IF NOT (Transfer.Mode = FIT_VFD_Transfer_Modes.Pause) AND NOT (Transfer.Mode = FIT_VFD_Transfer_Modes.Resume) THEN _w1 := Transfer.Mode; END_IF
Transfer.cONFIG.Mode_Memory := _w1;
IF Transfer.Mode = FIT_VFD_Transfer_Modes.Resume THEN _w2 := Transfer.Config.Mode_Memory; END_IF
Transfer.Mode := _w2;
Transfer.Status := SEL(False, SEL(BCV_Not_Ready, SEL(ACV_Not_Ready, SEL(Transfer.Mode=FIT_VFD_Transfer_Modes.Lock_Out, SEL(False, SEL(Complete, SEL(Transfer_Running, SEL(FIT.PLC_Reset, SEL(IDLE_Return, SEL(PAUSED, Transfer_status.IDLE, Transfer_status.Paused), Transfer_status.IDLE), Transfer_status.FIT_Reset), Transfer_status.Running), Transfer_status.Complete), Transfer_status.Complete), Transfer_status.LOCKED_OUT), Transfer_status.ACV_Not_Ready), Transfer_status.BCV_Not_Ready), Transfer_status.VFD_Not_Ready);
_w3 := Transfer.Mode = FIT_VFD_Transfer_Modes.Idle;
_w4 := True AND NOT (BCV.Status = eBCV_Status.A_Closed);
SR2(SET1 := _w3 AND _w4, RESET := NOT _w4); // SR
IF SR2.Q1 THEN _w5 := FIT_VFD_Transfer_Modes.Idle; END_IF
Transfer.Mode := _w5;
BCV_Not_Ready := _w3 AND _w4;
_w6 := 100 - (Transfer.Config.Target_Rate*Transfer.Config.FF);
Transfer.Current_Rate := SEL(Transfer.Config.Active, 0.0, FIT.Rate);
Transfer.Remaining_Time_S := REAL_TO_UDINT(SEL(Transfer_Running, 0.0, Transfer.Remaining_Volume/(Fit.Rate/60)));
_w7 := Transfer.Status = Transfer_Status.Complete;
_w8 := Transfer.Status = Transfer_Status.BCV_Not_Ready OR Transfer.Status = Transfer_Status.VFD_Not_Ready;
_w9 := Transfer_Status.IDLE = Transfer.Status OR False OR Transfer.Status = Transfer_Status.LOCKED_OUT;
_w10 := Transfer.Mode = FIT_VFD_Transfer_Modes.Pause;
PAUSED := _w10;
_w11 := Transfer.Mode = FIT_VFD_Transfer_Modes.IDLE;
_w12 := Complete OR Error OR _w11 OR _w10 OR False;
F_TRIG_0(CLK := Transfer_Running); // F_Trig
TP11(IN := NOT LockOut_Active AND _w12 AND BCV.PLC_CMD, PT := t#1s); // TP
BCV.PLC_CMD := SEL(F_TRIG_0.Q, BCV.PLC_CMD, False);
IDLE_Return := _w8 AND _w11;
SR_10(SET1 := FIT.Total<1, RESET := _w11); // SR
TON_10(IN := SR_10.Q1, PT := T#2s); // TON
FIT_Reset_Complete := TON_10.Q;
R_TRIG_0(CLK := _w11 OR TON_10.Q); // R_trig
_w13 := SEL(R_TRIG_0.Q, FIT.PLC_Reset, False);
_w14 := Transfer.Mode = FIT_VFD_Transfer_Modes.Batch;
_w15 := False OR False OR _w14;
Flow_Mode := _w15;
_w16 := _w15 AND FIT_Reset_Complete AND NOT Complete AND NOT Error AND NOT Time_Complete;
_w17 := _w16 OR (Transfer.Mode=FIT_VFD_Transfer_Modes.Passive);
FT_PIDW_1(
    IN := Transfer.Config.Target_Rate - FIT.Rate,
    KP := Transfer.Config.KP,
    TN := Transfer.Config.TN,
    TV := Transfer.Config.TV,
    LIM_L := 0,
    LIM_H := _w6,
    RST := NOT _w16); // BURKERT_OSCAT_BASIC.FT_PIDW
Transfer.Config.Motor_PCT := SEL(NOT Transfer_Running, LIMIT(0, 100, FT_PIDW_1.Y), 0.0);
Transfer.Config.Active := _w17;
Transfer_Running := _w17;
BCV.PLC_CMD := SEL(_w17, BCV.PLC_CMD, TRUE);
transfer.Remaining_Volume := SEL(_w16, Transfer.Config.Target_Volume, Transfer.Config.Target_Volume-fit.Total);
_w18 := _w14 AND FIT_Reset_Complete AND FIT.Total >= Transfer.Config.Target_Volume;
Batch_Complete := _w18;
RS_11(SET := Time_Complete OR _w18 OR False, RESET1 := _w11); // RS
Complete := RS_11.Q1;
_w19 := LOCK_OUT AND _w9 AND NOT RS_11.Q1;
F_TRIG_10(CLK := _w19); // F_Trig
IF F_TRIG_10.Q THEN _w20 := FIT_VFD_Transfer_Modes.Idle; END_IF
Transfer.Mode := _w20;
_w21 := _w19;
IF _w21 THEN _w22 := FIT_VFD_Transfer_Modes.Lock_Out; END_IF
LockOut_Active := _w21;
Transfer.Mode := _w22;
FIT.PLC_Reset := SEL(NOT SR_10.Q1 AND _w15 AND NOT _w18, _w13, True);
TON_12(IN := _w7, PT := T#30s); // TON
IF TON_12.Q THEN _w23 := FIT_VFD_Transfer_Modes.Idle; END_IF
Transfer.Mode := _w23;
Transfer.Current_Volume := SEL(Transfer.Config.Active, 0.0, FIT.Total);
// Transfer.Mode=FIT_VFD_Transfer_Modes.Passive: input not connected

END_FUNCTION_BLOCK

// 20 Program Organization Units/Transfer_BCV_VFD_FIT_UDFB
FUNCTION_BLOCK Transfer_BCV_VFD_FIT_UDFB
VAR_INPUT
	//Index:INT;
	LOCK_OUT:BOOL:=FALSE;
	
END_VAR
VAR_OUTPUT
END_VAR
VAR
	Paused:BOOL;
	Idle_return:BOOL;
	Transfer_Running:BOOL;
	Complete:BOOL;
	ACV_Not_Ready:BOOL;
	VFD_Not_Ready:BOOL;
	BCV_Not_Ready:BOOL;
	Time_Complete:BOOL;
	FIT_Reset_Complete:BOOL;
	Pump_Start:BOOL;
	Lockout_Active:BOOL;
	Error:BOOL;
	Flow_Mode:BOOL;
	Batch_Complete:BOOL;
	Enable_pump:BOOL;
	
	PID_CV:REAL;
	
	
	
	
	SR2: SR;
	TON_0: TON;
	CTRL_PID_1: BURKERT_OSCAT_BASIC.CTRL_PID;
	R_TRIG_0: R_trig;
	TON_10: TON;
	SR_10: SR;
	RS_11: RS;
	TON_12: TON;
	F_TRIG_10: F_Trig;
	TP11: TP;
	F_TRIG_0: F_Trig;
END_VAR

VAR_IN_OUT
	Transfer:FIT_VFD_Transfer_DUT;
	VFD:VFD_Vacon_DUT;
	BCV:BCV_DUT;
	FIT:FIT_DUT;
	
END_VAR
VAR // added by the converter: edge detectors and wires of the graphical bodies
    _w1, _w2, _w7, _w22, _w24 : ANY;
    _w3, _w4, _w5, _w6, _w8, _w9, _w10, _w11, _w12, _w13, _w14, _w15, _w16, _w17, _w18, _w19, _w20, _w21, _w23, _w25 : BOOL;
    _w26 : REAL;
END_VAR

IF NOT (Transfer.Mode = FIT_VFD_Transfer_Modes.Pause) AND NOT (Transfer.Mode = FIT_VFD_Transfer_Modes.Resume) THEN _w1 := Transfer.Mode; END_IF
Transfer.cONFIG.Mode_Memory := _w1;
IF Transfer.Mode = FIT_VFD_Transfer_Modes.Resume THEN _w2 := Transfer.Config.Mode_Memory; END_IF
Transfer.Mode := _w2;
Transfer.Status := SEL(VFD_Not_Ready, SEL(BCV_Not_Ready, SEL(ACV_Not_Ready, SEL(Transfer.Mode=FIT_VFD_Transfer_Modes.Lock_Out, SEL(False, SEL(Complete, SEL(Transfer_Running, SEL(FIT.PLC_Reset, SEL(IDLE_Return, SEL(PAUSED, Transfer_status.IDLE, Transfer_status.Paused), Transfer_status.IDLE), Transfer_status.FIT_Reset), Transfer_status.Running), Transfer_status.Complete), Transfer_status.Complete), Transfer_status.LOCKED_OUT), Transfer_status.ACV_Not_Ready), Transfer_status.BCV_Not_Ready), Transfer_status.VFD_Not_Ready);
_w3 := Transfer.Mode = FIT_VFD_Transfer_Modes.Idle;
_w4 := True AND NOT (BCV.Status = eBCV_Status.A_Closed);
BCV_Not_Ready := _w3 AND _w4;
_w5 := True AND NOT (VFD.MODE.eMode = VFD_Modes.Auto);
_w6 := _w4 OR _w5;
SR2(SET1 := _w3 AND _w6, RESET := NOT _w6); // SR
IF SR2.Q1 THEN _w7 := FIT_VFD_Transfer_Modes.Idle; END_IF
Transfer.Mode := _w7;
VFD_Not_Ready := _w3 AND _w5;
_w8 := Transfer.Status = Transfer_Status.Complete;
_w9 := Transfer.Status = Transfer_Status.BCV_Not_Ready OR Transfer.Status = Transfer_Status.VFD_Not_Ready;
_w10 := Transfer_Status.IDLE = Transfer.Status OR False OR Transfer.Status = Transfer_Status.LOCKED_OUT;
_w11 := Transfer.Mode = FIT_VFD_Transfer_Modes.Pause;
PAUSED := _w11;
_w12 := Transfer.Mode = FIT_VFD_Transfer_Modes.IDLE;
_w13 := Complete OR Error OR _w12 OR _w11;
_w14 := NOT Pump_Start OR _w13;
CTRL_PID_1(
    ACT := FIT.Rate,
    SET := Transfer.Config.Target_Rate,
    SUP := 0.0,
    OFS := Transfer.Config.Target_Rate * Transfer.Config.FF,
    M_I := 0.0,
    MAN := _w14,
    RST := _w14,
    KP := Transfer.Config.KP,
    TN := Transfer.Config.TN,
    TV := Transfer.Config.TV,
    LL := 0,
    LH := 100); // BURKERT_OSCAT_BASIC.CTRL_PID
PID_CV := CTRL_PID_1.Y;
TP11(IN := NOT LockOut_Active AND _w13, PT := t#5s); // TP
VFD.PLC_Run := SEL(TP11.Q, VFD.PLC_Run, FALSE);
VFD.PLC_CMD := SEL(TP11.Q, VFD.PLC_CMD, 0.0);
F_TRIG_0(CLK := TP11.Q); // F_Trig
BCV.PLC_CMD := SEL(F_TRIG_0.Q, BCV.PLC_CMD, False);
IDLE_Return := _w9 AND _w12;
SR_10(SET1 := FIT.Total<1, RESET := _w12); // SR
TON_10(IN := SR_10.Q1, PT := T#2s); // TON
FIT_Reset_Complete := TON_10.Q;
R_TRIG_0(CLK := _w12 OR TON_10.Q); // R_trig
_w15 := SEL(R_TRIG_0.Q, FIT.PLC_Reset, False);
_w16 := Transfer.Mode = FIT_VFD_Transfer_Modes.Batch;
_w17 := False OR False OR _w16;
Flow_Mode := _w17;
_w18 := _w17 AND FIT_Reset_Complete AND NOT Complete AND NOT Error AND NOT Time_Complete;
Transfer_Running := _w18;
transfer.Remaining_Volume := SEL(_w18, 0, Transfer.Config.Target_Volume-fit.Total);
_w19 := True AND _w18;
Enable_Pump := _w19;
BCV.PLC_CMD := SEL(_w19, BCV.PLC_CMD, TRUE);
_w20 := _w16 AND FIT_Reset_Complete AND FIT.Total >= Transfer.Config.Target_Volume;
Batch_Complete := _w20;
RS_11(SET := Time_Complete OR _w20 OR False, RESET1 := _w12); // RS
Complete := RS_11.Q1;
_w21 := LOCK_OUT AND _w10 AND NOT RS_11.Q1;
F_TRIG_10(CLK := _w21); // F_Trig
IF F_TRIG_10.Q THEN _w22 := FIT_VFD_Transfer_Modes.Idle; END_IF
Transfer.Mode := _w22;
_w23 := _w21;
IF _w23 THEN _w24 := FIT_VFD_Transfer_Modes.Lock_Out; END_IF
LockOut_Active := _w23;
Transfer.Mode := _w24;
FIT.PLC_Reset := SEL(NOT SR_10.Q1 AND _w17 AND NOT _w20, _w15, True);
_w25 := SEL(_w19, _w18, BCV.Status = eBCV_Status.A_Open);
Pump_Start := _w25;
_w26 := SEL(_w25, VFD.PLC_CMD, PID_CV);
Transfer.Config.Motor_PCT := _w26;
VFD.PLC_CMD := _w26;
VFD.PLC_Run := SEL(_w25, VFD.PLC_Run, PID_CV > 15);
TON_12(IN := _w8, PT := T#10s); // TON

END_FUNCTION_BLOCK

// 50 Functions/Alarm_Offset_Convert
FUNCTION Alarm_Offset_Convert : BOOL;
VAR_INPUT
	Config:cAlarm_Offsets;
	Alarm:REFERENCE TO cAlarm_Config;
END_VAR
VAR
END_VAR



Alarm.Setpoints.Alarm_Debounce:=Config.Alarm_Debounce;
Alarm.Setpoints.Warn_Debounce:=Config.Warn_Debounce;
Alarm.Setpoints.Hysteresis:=Config.Hysteresis;

Alarm.Setpoints.Hi_Hi_Alarm:=(COnfig.Target+Config.Hi_Hi_Alarm);
Alarm.Setpoints.Hi_Warn:=Config.Target+Config.Hi_Warn;
Alarm.Setpoints.Hi_Norm:=Config.Target+Config.Hi_Norm;
Alarm.Setpoints.Target:=Config.Target;
Alarm.Setpoints.Low_Norm:=Config.Target-Config.Low_Norm;
Alarm.Setpoints.Low_warn:=Config.Target-Config.Low_warn;
Alarm.Setpoints.Low_Low_Alarm:=Config.Target-Config.Low_Low_Alarm;


//IF Config.Target=0 THEN Alarm.Setpoints.Target:=(Alarm.Setpoints.Hi_Hi_Alarm+Alarm.Setpoints.Low_Low_Alarm)/2; END_IF;
IF Config.Hi_Norm=0 THEN Alarm.Setpoints.Hi_Norm:=Alarm.Setpoints.Target+(Alarm.Setpoints.Hi_Warn/2);END_IF
IF Config.Low_Norm=0 THEN Alarm.Setpoints.Low_Norm:=Alarm.Setpoints.Target+(Alarm.Setpoints.Low_warn/2);END_IF

END_FUNCTION

// 50 Functions/Alarm_Window_Convert
FUNCTION Alarm_Window_Convert : BOOL
VAR_INPUT
	Window: REFERENCE TO	 cAlarm_Window;
	Config:	REFERENCE TO	cAlarm_Config;
	
END_VAR
VAR
END_VAR

Config.Setpoints.Alarm_Debounce:=Window.Alarm_Delay;
Config.Setpoints.Warn_Debounce:=Window.Alarm_Delay/2;
Config.Setpoints.Hi_Hi_Alarm:= (Window.Target+Window.Alarm_Window);
Config.Setpoints.Hi_Warn:=(Window.Target+Window.Warn_Window);
Config.Setpoints.Low_warn:=(Window.Target-Window.Warn_Window);
Config.Setpoints.Low_Low_Alarm:=(Window.Target-Window.Alarm_Window);

END_FUNCTION

// 50 Functions/Anton_Parr_Deox
FUNCTION Anton_Parr_Deox : bool
VAR_INPUT
	Data:ARRAY[0..27] OF WORD;
END_VAR
VAR
END_VAR
VAR_OUTPUT
	C02_Vol:REAL;
	CO2_g_l_:REAL;
	CO2_bar:REAL;
	CO2_MPa:REAL;
	Temperature_C:REAL;
	Temperature_K:REAL;
	Temperature_F:REAL;
	Line_pressure_MPa:REAL;
	Days_to_next_maintenance:REAL;
	
	
	
	
END_VAR

END_FUNCTION

// 50 Functions/ASi_8694_Mapping
FUNCTION ASi_8694_Mapping : BOOL
VAR_INPUT
	Data_In:WORD;
	Setpoint:REAL;
END_VAR
VAR
END_VAR
VAR_OUTPUT
	Actual:REAL;
	Data_Out:word;
END_VAR

Actual := (INT_TO_REAL(WORD_TO_INT(Data_In))) / 100.0;
Data_Out := REAL_TO_WORD(Setpoint * 100.0);

END_FUNCTION

// 50 Functions/b8619_CND_FB
FUNCTION_BLOCK b8619_CND_FB
VAR_INPUT
	RX:POINTER TO BYTE;
END_VAR
VAR_OUTPUT
	Data:B8619_CND_DUT;
END_VAR
VAR
	Raw_ID:BYTE;
	Raw_Status:Byte;
END_VAR

raw_id:=rx[0];
	data.ID_Revision.0:=Raw_ID.0;
	data.ID_Revision.1:=Raw_id.1;
	Data.ID_Revision.2:=Raw_id.2;
	Data.ID_Revision.3:=Raw_id.3;
	
	Data.ID_Version.0:=Raw_id.4;
	Data.ID_Version.1:=Raw_ID.5;
	Data.ID_Version.2:=Raw_ID.6;
	Data.ID_Version.3:=Raw_ID.7;
raw_id:=rx[1];
	Data.ID_Slot.0:=Raw_ID.0;
	Data.ID_Slot.1:=Raw_ID.1;
	Data.ID_Slot.2:=Raw_ID.2;
	Data.ID_Slot.3:=Raw_ID.3;
	
	Data.ID_Type.0:=Raw_ID.4;
	Data.ID_Type.1:=Raw_ID.5;
	Data.ID_Type.2:=Raw_ID.6;
	Data.ID_Type.3:=Raw_ID.7;
	
Raw_Status:=RX[2];
	Data.Status_Link_Lost:=Raw_Status.0;
	Data.Status_Calibration_Lost:=Raw_Status.1;
	Data.Status_UserData_lost:=Raw_Status.2;
	Data.Status_Factory_Data_Lost:=Raw_Status.3;
	Data.Status_Probe_Error:=Raw_Status.4;
	Data.Status_Probe_Warning:=Raw_Status.6;
Raw_Status:=RX[3];
	Data.Status_Probe_Calibration	:=Raw_Status.0;
	Data.Status_Presence:=Raw_Status.7;

MEMUtils.MemCpy(pbyDest:=ADR(Data.Temp_Status) , pbySrc:=rx+4 , dwSize:=2 );
MEMUtils.MemCpy(pbyDest:=ADR(Data.CND_Status) , pbySrc:=rx+6 , dwSize:=2 );
MEMUtils.MemCpy(pbyDest:=ADR(Data.RTD)+2 , pbySrc:=rx+12 , dwSize:=2 );
MEMUtils.MemCpy(pbyDest:=ADR(Data.RTD) , pbySrc:=rx+14 , dwSize:=2 );

MEMUtils.MemCpy(pbyDest:=ADR(Data.Temperature)+2 , pbySrc:=rx+16 , dwSize:=2 );
MEMUtils.MemCpy(pbyDest:=ADR(Data.Temperature) , pbySrc:=rx+18 , dwSize:=2 );
MEMUtils.MemCpy(pbyDest:=ADR(Data.Conductivity)+2 , pbySrc:=rx+20 , dwSize:=2 );
MEMUtils.MemCpy(pbyDest:=ADR(Data.Conductivity) , pbySrc:=rx+22 , dwSize:=2 );
MEMUtils.MemCpy(pbyDest:=ADR(Data.Resistivity)+2 , pbySrc:=rx+24 , dwSize:=2 );
MEMUtils.MemCpy(pbyDest:=ADR(Data.Resistivity) , pbySrc:=rx+26 , dwSize:=2 );
MEMUtils.MemCpy(pbyDest:=ADR(Data.TDS)+2 , pbySrc:=rx+28 , dwSize:=2 );
MEMUtils.MemCpy(pbyDest:=ADR(Data.TDS) , pbySrc:=rx+30 , dwSize:=2 );
MEMUtils.MemCpy(pbyDest:=ADR(Data.Concentration)+2 , pbySrc:=rx+32 , dwSize:=2 );
MEMUtils.MemCpy(pbyDest:=ADR(Data.Concentration) , pbySrc:=rx+34 , dwSize:=2 );

END_FUNCTION_BLOCK

// 50 Functions/B8619_Input_FB
FUNCTION_BLOCK B8619_Input_FB
VAR_INPUT
	RX:POINTER TO BYTE;
END_VAR
VAR_OUTPUT
	Data:B8619_inputs_DUT;
END_VAR
VAR
	Raw_ID:BYTE;
	Raw_Status:Byte;
END_VAR

raw_id:=rx[0];
	data.ID_Revision.0:=Raw_ID.0;
	data.ID_Revision.1:=Raw_id.1;
	Data.ID_Revision.2:=Raw_id.2;
	Data.ID_Revision.3:=Raw_id.3;
	
	Data.ID_Version.0:=Raw_id.4;
	Data.ID_Version.1:=Raw_ID.5;
	Data.ID_Version.2:=Raw_ID.6;
	Data.ID_Version.3:=Raw_ID.7;
raw_id:=rx[1];
	Data.ID_Slot.0:=Raw_ID.0;
	Data.ID_Slot.1:=Raw_ID.1;
	Data.ID_Slot.2:=Raw_ID.2;
	Data.ID_Slot.3:=Raw_ID.3;
	
	Data.ID_Type.0:=Raw_ID.4;
	Data.ID_Type.1:=Raw_ID.5;
	Data.ID_Type.2:=Raw_ID.6;
	Data.ID_Type.3:=Raw_ID.7;
	
Raw_Status:=RX[2];
	Data.Status_Link_Lost:=Raw_Status.0;
	Data.Status_Calibration_Lost:=Raw_Status.1;
	Data.Status_UserData_lost:=Raw_Status.2;
	Data.Status_Factory_Data_Lost:=Raw_Status.3;
	Data.Status_time_lost:=Raw_Status.4;
	Data.Status_Warning:=Raw_Status.6;
Raw_Status:=RX[3];
	Data.Status_Memory_Issue	:=Raw_Status.0;
	Data.Status_Presence:=Raw_Status.7;
	

MEMUtils.MemCpy(pbyDest:=ADR(Data.DI1_Status) , pbySrc:=rx+4 , dwSize:=2);
MEMUtils.MemCpy(pbyDest:=ADR(Data.DI2_Status) , pbySrc:=rx+6 , dwSize:=2);
MEMUtils.MemCpy(pbyDest:=ADR(Data.AI1_Status) , pbySrc:=rx+8 , dwSize:=2);
MEMUtils.MemCpy(pbyDest:=ADR(Data.AI2_Status) , pbySrc:=rx+10 , dwSize:=2);

MEMUtils.MemCpy(pbyDest:=ADR(Data.DI1_Hz)+2 , pbySrc:=rx+12 , dwSize:=2);
MEMUtils.MemCpy(pbyDest:=ADR(Data.DI1_Hz) , pbySrc:=rx+14 , dwSize:=2);

MEMUtils.MemCpy(pbyDest:=ADR(Data.DI1_Flow)+2 , pbySrc:=rx+16 , dwSize:=2);
MEMUtils.MemCpy(pbyDest:=ADR(Data.DI1_Flow) , pbySrc:=rx+18 , dwSize:=2);

MEMUtils.MemCpy(pbyDest:=ADR(Data.DI1_Total_A)+2 , pbySrc:=rx+20 , dwSize:=2);
MEMUtils.MemCpy(pbyDest:=ADR(Data.DI1_Total_A) , pbySrc:=rx+22 , dwSize:=2);

MEMUtils.MemCpy(pbyDest:=ADR(Data.DI1_Total_B)+2 , pbySrc:=rx+24 , dwSize:=2);
MEMUtils.MemCpy(pbyDest:=ADR(Data.DI1_Total_B) , pbySrc:=rx+26 , dwSize:=2);	

MEMUtils.MemCpy(pbyDest:=ADR(Data.DI2_Hz)+2 , pbySrc:=rx+28 , dwSize:=2);
MEMUtils.MemCpy(pbyDest:=ADR(Data.DI2_Hz) , pbySrc:=rx+30 , dwSize:=2);

MEMUtils.MemCpy(pbyDest:=ADR(Data.DI2_Flow)+2 , pbySrc:=rx+32 , dwSize:=2);
MEMUtils.MemCpy(pbyDest:=ADR(Data.DI2_Flow) , pbySrc:=rx+34 , dwSize:=2);

MEMUtils.MemCpy(pbyDest:=ADR(Data.DI2_Total_A)+2 , pbySrc:=rx+36 , dwSize:=2);
MEMUtils.MemCpy(pbyDest:=ADR(Data.DI2_Total_A) , pbySrc:=rx+38 , dwSize:=2);

MEMUtils.MemCpy(pbyDest:=ADR(Data.DI2_Total_B)+2 , pbySrc:=rx+40 , dwSize:=2);
MEMUtils.MemCpy(pbyDest:=ADR(Data.DI2_Total_B) , pbySrc:=rx+42 , dwSize:=2);	

MEMUtils.MemCpy(pbyDest:=ADR(Data.AI1_Raw)+2 , pbySrc:=rx+44 , dwSize:=2);
MEMUtils.MemCpy(pbyDest:=ADR(Data.AI1_Raw) , pbySrc:=rx+46 , dwSize:=2);

MEMUtils.MemCpy(pbyDest:=ADR(Data.AI1_EU)+2 , pbySrc:=rx+48 , dwSize:=2);
MEMUtils.MemCpy(pbyDest:=ADR(Data.AI1_EU) , pbySrc:=rx+50 , dwSize:=2);

MEMUtils.MemCpy(pbyDest:=ADR(Data.AI2_Raw)+2 , pbySrc:=rx+52 , dwSize:=2);
MEMUtils.MemCpy(pbyDest:=ADR(Data.AI2_Raw) , pbySrc:=rx+54 , dwSize:=2);

MEMUtils.MemCpy(pbyDest:=ADR(Data.AI2_EU)+2 , pbySrc:=rx+56 , dwSize:=2);
MEMUtils.MemCpy(pbyDest:=ADR(Data.AI2_EU) , pbySrc:=rx+58 , dwSize:=2);

END_FUNCTION_BLOCK

// 50 Functions/B8619_Main_FB
FUNCTION_BLOCK B8619_Main_FB
VAR_INPUT
	RX:POINTER TO BYTE;
END_VAR
VAR_OUTPUT
	Data:B8619_Main_DUT;
END_VAR
VAR
	Raw_ID:BYTE;
	Raw_Status:Byte;
END_VAR

raw_id:=rx[0];
	data.ID_Revision.0:=Raw_ID.0;
	data.ID_Revision.1:=Raw_id.1;
	Data.ID_Revision.2:=Raw_id.2;
	Data.ID_Revision.3:=Raw_id.3;
	
	Data.ID_Version.0:=Raw_id.4;
	Data.ID_Version.1:=Raw_ID.5;
	Data.ID_Version.2:=Raw_ID.6;
	Data.ID_Version.3:=Raw_ID.7;
raw_id:=rx[1];
	Data.ID_Slot.0:=Raw_ID.0;
	Data.ID_Slot.1:=Raw_ID.1;
	Data.ID_Slot.2:=Raw_ID.2;
	Data.ID_Slot.3:=Raw_ID.3;
	
	Data.ID_Type.0:=Raw_ID.4;
	Data.ID_Type.1:=Raw_ID.5;
	Data.ID_Type.2:=Raw_ID.6;
	Data.ID_Type.3:=Raw_ID.7;
	
Raw_Status:=RX[2];
	Data.Status_Link_Lost:=Raw_Status.0;
	Data.Status_Calibration_Lost:=Raw_Status.1;
	Data.Status_UserData_lost:=Raw_Status.2;
	Data.Status_Factory_Data_Lost:=Raw_Status.3;
	Data.Status_time_lost:=Raw_Status.4;
	Data.Status_Warning:=Raw_Status.6;
Raw_Status:=RX[3];
	Data.Status_Memory_Issue	:=Raw_Status.0;
	Data.Status_Presence:=Raw_Status.7;
	
MEMUtils.MemCpy(pbyDest:=ADR(Data.M1_M3_Status) , pbySrc:=rx+4 , dwSize:=2 );
MEMUtils.MemCpy(pbyDest:=ADR(Data.M4_M6_Status) , pbySrc:=rx+6 , dwSize:=2);
MEMUtils.MemCpy(pbyDest:=ADR(Data.System_Switch) , pbySrc:=rx+8 , dwSize:=2);
MEMUtils.MemCpy(pbyDest:=ADR(Data.DI1_Status) , pbySrc:=rx+10 , dwSize:=2);
MEMUtils.MemCpy(pbyDest:=ADR(Data.DI2_Status) , pbySrc:=rx+12 , dwSize:=2);
MEMUtils.MemCpy(pbyDest:=ADR(Data.DO1) , pbySrc:=rx+14 , dwSize:=2);
MEMUtils.MemCpy(pbyDest:=ADR(Data.DO2) , pbySrc:=rx+16 , dwSize:=2);

MEMUtils.MemCpy(pbyDest:=ADR(Data.AO1) , pbySrc:=rx+18 , dwSize:=2);
MEMUtils.MemCpy(pbyDest:=ADR(Data.AO1)+2 , pbySrc:=rx+20 , dwSize:=2);

MEMUtils.MemCpy(pbyDest:=ADR(Data.AO2) , pbySrc:=rx+22 , dwSize:=2);
MEMUtils.MemCpy(pbyDest:=ADR(Data.AO2)+2 , pbySrc:=rx+24 , dwSize:=2);

MEMUtils.MemCpy(pbyDest:=ADR(Data.DI1_Hz) , pbySrc:=rx+26 , dwSize:=2);
MEMUtils.MemCpy(pbyDest:=ADR(Data.DI1_Hz)+2 , pbySrc:=rx+28 , dwSize:=2);

MEMUtils.MemCpy(pbyDest:=ADR(Data.DI1_Flow) , pbySrc:=rx+30 , dwSize:=2);
MEMUtils.MemCpy(pbyDest:=ADR(Data.DI1_Flow)+2 , pbySrc:=rx+32 , dwSize:=2);

MEMUtils.MemCpy(pbyDest:=ADR(Data.DI1_Total_A) , pbySrc:=rx+34 , dwSize:=2);
MEMUtils.MemCpy(pbyDest:=ADR(Data.DI1_Total_A)+2 , pbySrc:=rx+36 , dwSize:=2);

MEMUtils.MemCpy(pbyDest:=ADR(Data.DI1_Total_B) , pbySrc:=rx+38 , dwSize:=2);
MEMUtils.MemCpy(pbyDest:=ADR(Data.DI1_Total_B)+2 , pbySrc:=rx+40 , dwSize:=2);	

MEMUtils.MemCpy(pbyDest:=ADR(Data.DI2_Hz) , pbySrc:=rx+42 , dwSize:=2);
MEMUtils.MemCpy(pbyDest:=ADR(Data.DI2_Hz)+2 , pbySrc:=rx+44 , dwSize:=2);

MEMUtils.MemCpy(pbyDest:=ADR(Data.DI2_Flow) , pbySrc:=rx+46 , dwSize:=2);
MEMUtils.MemCpy(pbyDest:=ADR(Data.DI2_Flow)+2 , pbySrc:=rx+48 , dwSize:=2);

MEMUtils.MemCpy(pbyDest:=ADR(Data.DI2_Total_A) , pbySrc:=rx+50 , dwSize:=2);
MEMUtils.MemCpy(pbyDest:=ADR(Data.DI2_Total_A)+2 , pbySrc:=rx+52 , dwSize:=2);

MEMUtils.MemCpy(pbyDest:=ADR(Data.DI2_Total_B) , pbySrc:=rx+54 , dwSize:=2);
MEMUtils.MemCpy(pbyDest:=ADR(Data.DI2_Total_B)+2 , pbySrc:=rx+56 , dwSize:=2);

END_FUNCTION_BLOCK

// 50 Functions/b8619_PH_ORP_FB
FUNCTION_BLOCK b8619_PH_ORP_FB
VAR_INPUT
	RX:POINTER TO BYTE;
END_VAR
VAR_OUTPUT
	Data:B8619_PH_DUT;
END_VAR
VAR
	Raw_ID:BYTE;
	Raw_Status:Byte;
END_VAR

raw_id:=rx[0];
	data.ID_Revision.0:=Raw_ID.0;
	data.ID_Revision.1:=Raw_id.1;
	Data.ID_Revision.2:=Raw_id.2;
	Data.ID_Revision.3:=Raw_id.3;
	
	Data.ID_Version.0:=Raw_id.4;
	Data.ID_Version.1:=Raw_ID.5;
	Data.ID_Version.2:=Raw_ID.6;
	Data.ID_Version.3:=Raw_ID.7;
raw_id:=rx[1];
	Data.ID_Slot.0:=Raw_ID.0;
	Data.ID_Slot.1:=Raw_ID.1;
	Data.ID_Slot.2:=Raw_ID.2;
	Data.ID_Slot.3:=Raw_ID.3;
	
	Data.ID_Type.0:=Raw_ID.4;
	Data.ID_Type.1:=Raw_ID.5;
	Data.ID_Type.2:=Raw_ID.6;
	Data.ID_Type.3:=Raw_ID.7;
	
Raw_Status:=RX[2];
	Data.Status_Link_Lost:=Raw_Status.0;
	Data.Status_Calibration_Lost:=Raw_Status.1;
	Data.Status_UserData_lost:=Raw_Status.2;
	Data.Status_Factory_Data_Lost:=Raw_Status.3;
	Data.Status_Probe_Error:=Raw_Status.4;
	Data.Status_Probe_Warning:=Raw_Status.6;
Raw_Status:=RX[3];
	Data.Status_Probe_Calibration	:=Raw_Status.0;
	Data.Status_Presence:=Raw_Status.7;

MEMUtils.MemCpy(pbyDest:=ADR(Data.Temp_Status) , pbySrc:=ADR(rx)+4 , dwSize:=2 );
MEMUtils.MemCpy(pbyDest:=ADR(Data.PH_Status) , pbySrc:=ADR(rx)+6 , dwSize:=2 );
MEMUtils.MemCpy(pbyDest:=ADR(Data.RTD)+2 , pbySrc:=ADR(rx)+12 , dwSize:=2 );
MEMUtils.MemCpy(pbyDest:=ADR(Data.RTD) , pbySrc:=ADR(rx)+14 , dwSize:=2 );

MEMUtils.MemCpy(pbyDest:=ADR(Data.Temperature)+2 , pbySrc:=ADR(rx)+16 , dwSize:=2 );
MEMUtils.MemCpy(pbyDest:=ADR(Data.Temperature) , pbySrc:=ADR(rx)+18 , dwSize:=2 );
MEMUtils.MemCpy(pbyDest:=ADR(Data.mv_PH)+2 , pbySrc:=ADR(rx)+20 , dwSize:=2 );
MEMUtils.MemCpy(pbyDest:=ADR(Data.mv_PH) , pbySrc:=ADR(rx)+22 , dwSize:=2 );
MEMUtils.MemCpy(pbyDest:=ADR(Data.mv_ORP)+2 , pbySrc:=ADR(rx)+24 , dwSize:=2 );
MEMUtils.MemCpy(pbyDest:=ADR(Data.mv_ORP) , pbySrc:=ADR(rx)+26 , dwSize:=2 );
MEMUtils.MemCpy(pbyDest:=ADR(Data.PH)+2 , pbySrc:=ADR(rx)+28 , dwSize:=2 );
MEMUtils.MemCpy(pbyDest:=ADR(Data.PH) , pbySrc:=ADR(rx)+30 , dwSize:=2 );
MEMUtils.MemCpy(pbyDest:=ADR(Data.Impedance_Glass)+2 , pbySrc:=ADR(rx)+32 , dwSize:=2 );
MEMUtils.MemCpy(pbyDest:=ADR(Data.Impedance_Glass) , pbySrc:=ADR(rx)+34 , dwSize:=2 );
MEMUtils.MemCpy(pbyDest:=ADR(Data.Impedance_Ref)+2 , pbySrc:=ADR(rx)+36 , dwSize:=2 );
MEMUtils.MemCpy(pbyDest:=ADR(Data.Impedance_Ref) , pbySrc:=ADR(rx)+38 , dwSize:=2 );

END_FUNCTION_BLOCK

// 50 Functions/Build_ORF_Index
FUNCTION Build_ORF_Index : DWORD
VAR_INPUT
	Index:WORD;
	SubIndex:BYTE;
	Node:BYTE;
	Write:BOOL;
END_VAR
VAR
	uORF:Bytes_Dword;
END_VAR

uORF.tWord[0]:=Index;
uORF.tByte[3]:=SubIndex;
IF Write THEN
	uorf.tByte[2]:=node+16#80;
ELSE
	uorf.tByte[2]:=node;
END_IF;

Build_ORF_Index:=uORF.tDword;

END_FUNCTION

// 50 Functions/Contactor_Control_FB
FUNCTION Contactor_Control_FB : BOOL
VAR_INPUT
	Index:INT;
	Allow_Reverse:BOOL;
	Inhibit_FWD:BOOL:=FALSE;
	Inhibit_Rev:BOOL:=FALSE;
END_VAR
VAR_OUTPUT
	Q_FWD:BOOL;
	Q_REV:Bool;
END_VAR
VAR
	//F_TRIG_0: F_trig;
	TP_0: TP;
	F_TRIG_1: F_trig;
	TP_1: TP;
END_VAR
VAR // added by the converter: edge detectors and wires of the graphical bodies
    _w1, _w2, _w4, _w5, _w6, _w7, _w8, _w10, _w11, _w12 : BOOL;
    _w3, _w9 : ANY;
END_VAR

_w1 := GVL.BH_Contactor[Index].Mode = Contactor_Modes.Auto;
_w2 := _w1 AND GVL.BH_Contactor[Index].PLC_CMD_FWD;
_w3 := SEL(_w2, Contactor_Status.OFF, Contactor_Status.Auto_FWD);
_w4 := GVL.BH_Contactor[Index].Mode = Contactor_Modes.Fwd;
TP_1(IN := GVL.BH_Contactor[Index].Mode = Contactor_Modes.Bump_FWD, PT := T#1s); // TP
_w5 := _w4 OR TP_1.Q;
_w6 := _w2 OR _w5;
_w7 := _w6 AND NOT Inhibit_FWD;
GVL.BH_Contactor[Index].Q1 := _w7;
Q_FWD := _w7;
_w8 := _w1 AND GVL.BH_Contactor[Index].PLC_CMD_Rev;
_w9 := SEL(_w8, SEL(_w5, _w3, Contactor_Status.Manual_FWD), Contactor_Status.Auto_Rev);
_w10 := GVL.BH_Contactor[Index].Mode = Contactor_Modes.Rev;
TP_0(IN := GVL.BH_Contactor[Index].Mode = Contactor_Modes.Bump_REV, PT := T#1s); // TP
_w11 := _w10 OR TP_0.Q;
GVL.BH_Contactor[Index].Status := SEL(_w11, _w9, Contactor_Status.Manual_Rev);
_w12 := (NOT _w6 AND (_w8 OR _w11) AND Allow_Reverse) AND NOT Inhibit_REV;
Q_Rev := _w12;
GVL.BH_Contactor[Index].Q2 := _w12;
F_TRIG_1(CLK := TP_1.Q OR TP_0.Q); // F_trig
GVL.BH_Contactor[Index].Mode := SEL(F_TRIG_1.Q, GVL.BH_Contactor[Index].Mode, Contactor_Modes.Disabled);

END_FUNCTION

// 50 Functions/DaySeconds
FUNCTION DaySeconds : UDINT
VAR_INPUT
	Hour:UINT;
	Minute:UINT;
	Second:UINT;
END_VAR
VAR
END_VAR

(* body of a kind this reader does not render *)

END_FUNCTION

// 50 Functions/Find_Real_In_Array
FUNCTION Find_Real_In_Array 
VAR_INPUT
   key : REAL;
END_VAR
VAR_IN_OUT
   arr : ARRAY [*] OF REAL;
END_VAR
VAR_OUTPUT
	   out1 : INT;
   		out2 : INT;
END_VAR
VAR
   size : DINT;
   i: INT;
   j: INT;
   middle: INT;
END_VAR

size := UPPER_BOUND(arr,1);
IF key <= arr[0] THEN
   out1 := 0;
   out2 := 0;
   RETURN;
END_IF
IF key >= arr[size] THEN
   out1 := TO_INT(size);
   out2 := TO_INT(size);
   RETURN;
END_IF
i := 0;
j := TO_INT(size);
middle := 0;
WHILE (i < j) DO
   
   middle := (i+j)/2;
   IF key = arr[middle] THEN
       out1 := middle;
       out2 := middle;
       RETURN;
   END_IF
   
   IF key < arr[middle] THEN
      
      IF (middle > 0) AND (key > arr[middle - 1]) THEN
         
         IF key < 0 THEN
             out1 := middle - 1;
             out2 := middle;
         ELSE
             out1 := middle;
             out2 := middle - 1;
         END_IF
         RETURN;
      END_IF
      
      j := middle;
         
   ELSE
      
      IF (middle < size ) AND (key < arr[middle + 1]) THEN
          out1 := middle;
          out2 := middle + 1;
          RETURN;
      END_IF
 
      i := middle + 1;
      
   END_IF
END_WHILE

END_FUNCTION

// 50 Functions/FindClosestIndex
FUNCTION FindClosestIndex : INT
VAR_INPUT
    TargetValue : REAL;
    Increment : REAL;
    MaxIndex : INT;
END_VAR
VAR
    ClosestIndex : INT;
    i : INT;
END_VAR



ClosestIndex := 0;
FOR i := 0 TO MaxIndex DO
    IF ABS((i * Increment) - TargetValue) < ABS((ClosestIndex * Increment) - TargetValue) THEN
        ClosestIndex := i;
    END_IF
END_FOR

FindClosestIndex := ClosestIndex;

END_FUNCTION

// 50 Functions/FindClosestIndexSorted
FUNCTION FindClosestIndexSorted : INT
VAR_INPUT
    ArrayIn: ARRAY[*] OF REAL; // Dynamic array size
    TargetValue: REAL;
END_VAR
VAR
   Low: INT := 0;
    High: INT := TO_INT(UPPER_BOUND(ArrayIn, 1));
    Mid: INT;
    ClosestIndex: INT := 0;
    ClosestDifference: REAL := ABS(ArrayIn[0] - TargetValue);
    CurrentDifference: REAL;
END_VAR


WHILE Low <= High DO
	Mid := (Low + High) / 2;

	// Calculate the difference for the current midpoint
	CurrentDifference := ABS(ArrayIn[Mid] - TargetValue);

	// Update closest index if this midpoint is closer
	IF CurrentDifference < ClosestDifference THEN
		ClosestDifference := CurrentDifference;
		ClosestIndex := Mid;
	END_IF

	// Adjust search bounds based on target value
	IF ArrayIn[Mid] < TargetValue THEN
		Low := Mid + 1;
	ELSE
		High := Mid - 1;
	END_IF
END_WHILE

FindClosestIndexSorted := ClosestIndex;

END_FUNCTION

// 50 Functions/Calculators/MidPoint
FUNCTION MidPoint : REAL
VAR_INPUT
	A:REAL;
	B:REAL;
END_VAR
VAR
END_VAR

IF A<B THEN
	MidPoint:=(A+( (B-A)/2));
ELSE
	Midpoint:=(B+( (A-B)/2));
END_IF;

END_FUNCTION

// 50 Functions/FlowWave_Mapping
FUNCTION FlowWave_Mapping : cFLOWave_DUT
VAR_INPUT
	RX:ARRAY[0..17] OF WORD;
END_VAR
VAR
END_VAR

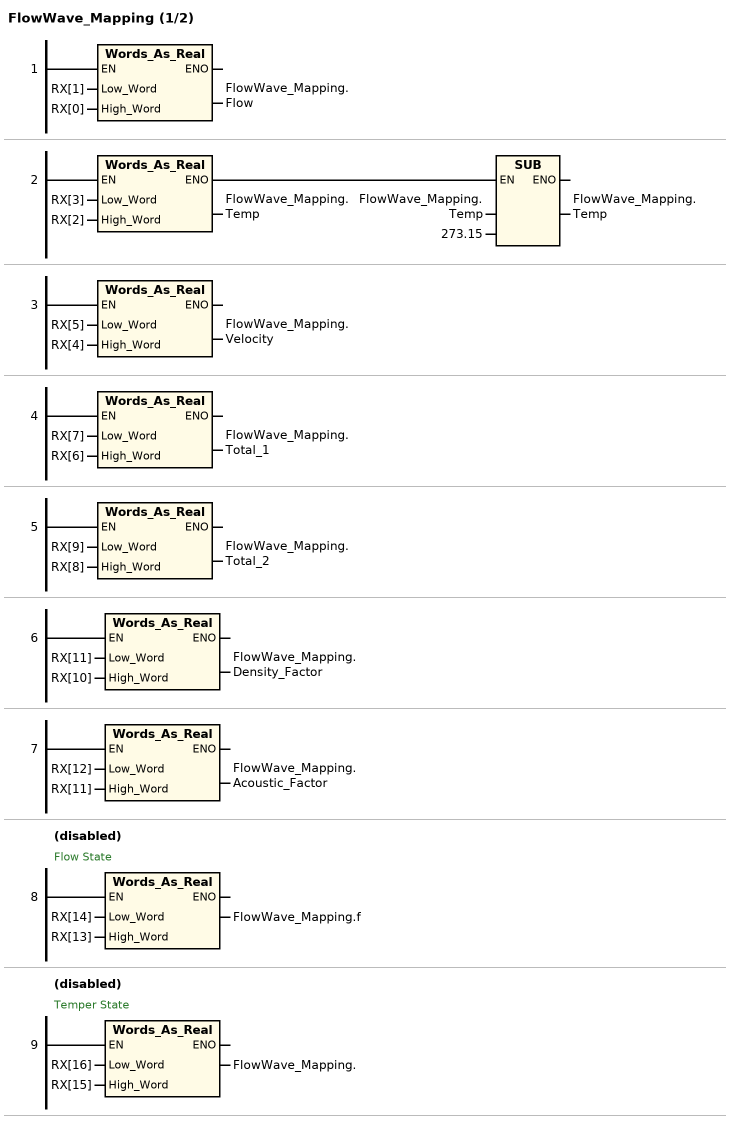
// NETWORK 1
FlowWave_Mapping.Flow := Words_As_Real(Low_Word := RX[1], High_Word := RX[0]);

// NETWORK 2
FlowWave_Mapping.Temp := Words_As_Real(Low_Word := RX[3], High_Word := RX[2]);
FlowWave_Mapping.Temp := FlowWave_Mapping.Temp - 273.15;

// NETWORK 3
FlowWave_Mapping.Velocity := Words_As_Real(Low_Word := RX[5], High_Word := RX[4]);

// NETWORK 4
FlowWave_Mapping.Total_1 := Words_As_Real(Low_Word := RX[7], High_Word := RX[6]);

// NETWORK 5
FlowWave_Mapping.Total_2 := Words_As_Real(Low_Word := RX[9], High_Word := RX[8]);

// NETWORK 6
FlowWave_Mapping.Density_Factor := Words_As_Real(Low_Word := RX[11], High_Word := RX[10]);

// NETWORK 7
FlowWave_Mapping.Acoustic_Factor := Words_As_Real(Low_Word := RX[12], High_Word := RX[11]);

// NETWORK 8 (disabled)
// Flow State
// FlowWave_Mapping.f := Words_As_Real(Low_Word := RX[14], High_Word := RX[13]);

// NETWORK 9 (disabled)
// Temper State
// FlowWave_Mapping. := Words_As_Real(Low_Word := RX[16], High_Word := RX[15]);

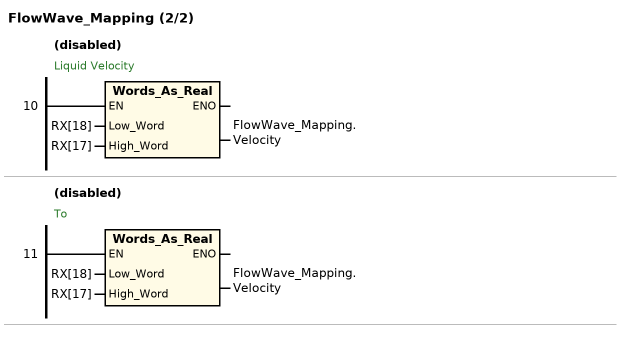
// NETWORK 10 (disabled)
// Liquid Velocity
// FlowWave_Mapping.Velocity := Words_As_Real(Low_Word := RX[18], High_Word := RX[17]);

// NETWORK 11 (disabled)
// To
// FlowWave_Mapping.Velocity := Words_As_Real(Low_Word := RX[18], High_Word := RX[17]);

END_FUNCTION

// 50 Functions/fNord_Control_Word
FUNCTION fNord_Control_Word : UINT
VAR_INPUT
	Control:cNord_Control_Word;
END_VAR
VAR
END_VAR

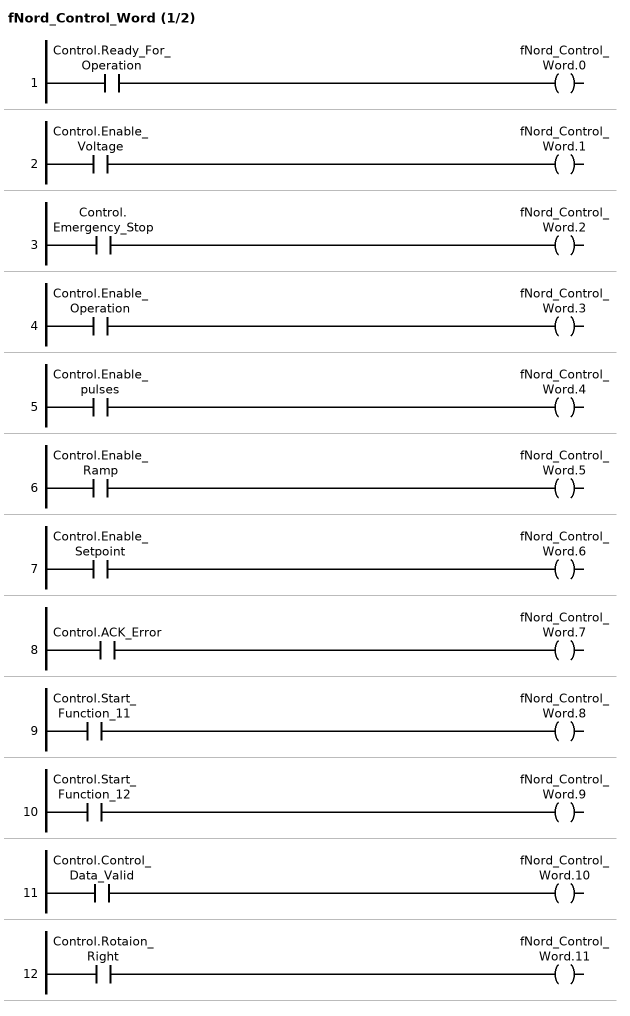
// NETWORK 1
fNord_Control_Word.0 := Control.Ready_For_Operation;

// NETWORK 2
fNord_Control_Word.1 := Control.Enable_Voltage;

// NETWORK 3
fNord_Control_Word.2 := Control.Emergency_Stop;

// NETWORK 4
fNord_Control_Word.3 := Control.Enable_Operation;

// NETWORK 5
fNord_Control_Word.4 := Control.Enable_pulses;

// NETWORK 6
fNord_Control_Word.5 := Control.Enable_Ramp;

// NETWORK 7
fNord_Control_Word.6 := Control.Enable_Setpoint;

// NETWORK 8
fNord_Control_Word.7 := Control.ACK_Error;

// NETWORK 9
fNord_Control_Word.8 := Control.Start_Function_11;

// NETWORK 10
fNord_Control_Word.9 := Control.Start_Function_12;

// NETWORK 11
fNord_Control_Word.10 := Control.Control_Data_Valid;

// NETWORK 12
fNord_Control_Word.11 := Control.Rotaion_Right;

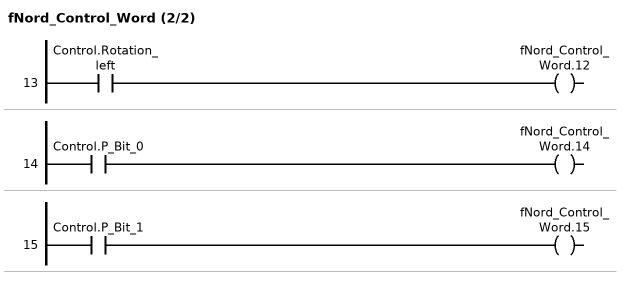
// NETWORK 13
fNord_Control_Word.12 := Control.Rotation_left;

// NETWORK 14
fNord_Control_Word.14 := Control.P_Bit_0;

// NETWORK 15
fNord_Control_Word.15 := Control.P_Bit_1;

END_FUNCTION

// 50 Functions/fNord_Status_Mapping
FUNCTION fNord_Status_Mapping : BOOL
VAR_INPUT
	Raw:UINT;
END_VAR
VAR
END_VAR
VAR_OUTPUT
	Status:cNord_Status;
END_VAR

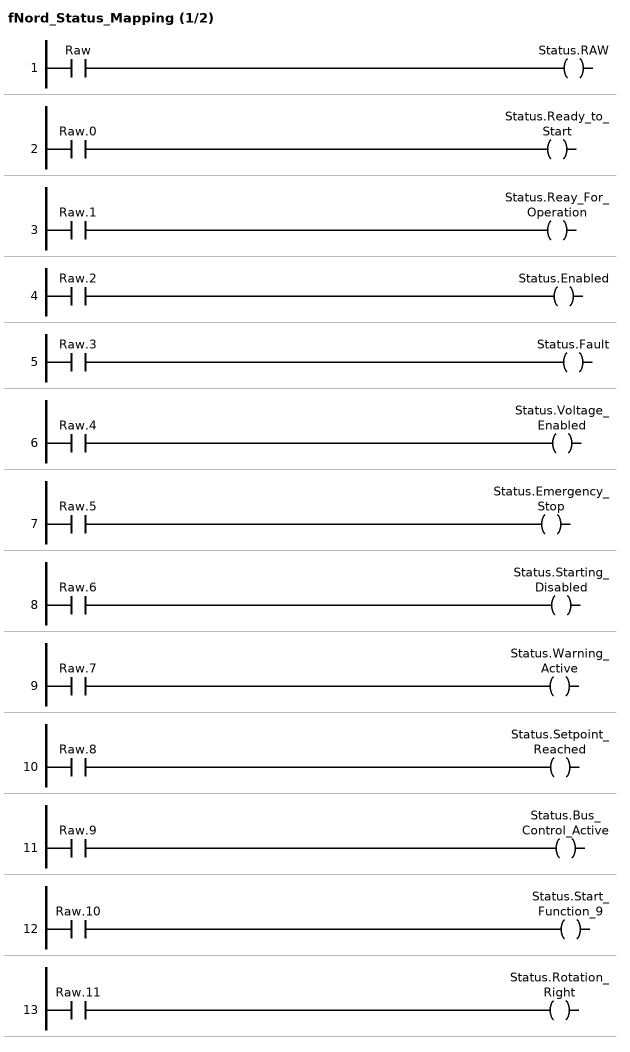
// NETWORK 1
Status.RAW := Raw;

// NETWORK 2
Status.Ready_to_Start := Raw.0;

// NETWORK 3
Status.Reay_For_Operation := Raw.1;

// NETWORK 4
Status.Enabled := Raw.2;

// NETWORK 5
Status.Fault := Raw.3;

// NETWORK 6
Status.Voltage_Enabled := Raw.4;

// NETWORK 7
Status.Emergency_Stop := Raw.5;

// NETWORK 8
Status.Starting_Disabled := Raw.6;

// NETWORK 9
Status.Warning_Active := Raw.7;

// NETWORK 10
Status.Setpoint_Reached := Raw.8;

// NETWORK 11
Status.Bus_Control_Active := Raw.9;

// NETWORK 12
Status.Start_Function_9 := Raw.10;

// NETWORK 13
Status.Rotation_Right := Raw.11;

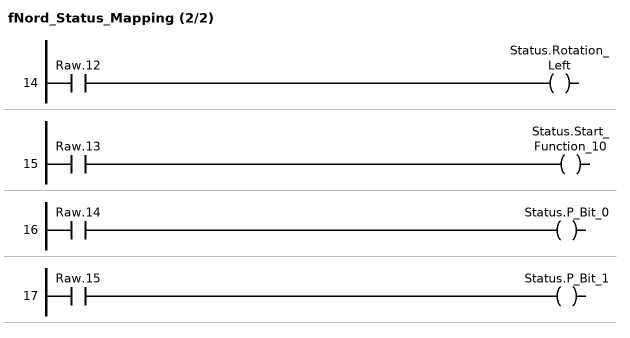
// NETWORK 14
Status.Rotation_Left := Raw.12;

// NETWORK 15
Status.Start_Function_10 := Raw.13;

// NETWORK 16
Status.P_Bit_0 := Raw.14;

// NETWORK 17
Status.P_Bit_1 := Raw.15;

END_FUNCTION

// 50 Functions/Tempered_Flow_Calculator
FUNCTION Tempered_Flow_Calculator : Bool
VAR_INPUT
	CT:REAL;
	HT:REAL;
	Required_Flow:REAL;
	Required_Temperature:REAL;
END_VAR
VAR_OUTPUT
	Hot_Flow:REAL;
	Cold_Flow:REAL;
END_VAR
VAR
END_VAR


 

Hot_Flow:=  Required_Flow *( (Required_Temperature-CT) / (HT-CT));
Cold_Flow:=	Required_Flow - Hot_Flow;

END_FUNCTION

// 50 Functions/Tempered_Look_UP
FUNCTION Tempered_Look_UP : Bool
VAR_INPUT
	Data:Tempered_Data;
	
END_VAR

VAR_OUTPUT
	FlowIndex, TempIndex : INT;

	
END_VAR
VAR
	
    FlowIncrement, TempIncrement : REAL;
END_VAR



// Assign values to the increments and target values

// Find the closest indices
FlowIndex := FindClosestIndex(Data.TargetFlow, Data.FlowIncrement, 20);
TempIndex := FindClosestIndex(Data.TargetTemperature, Data.TempIncrement, 20);

// Retrieve the KV values from the array
Data.CW1_KV := Data.Temperature[TempIndex][FlowIndex].CW1_KV;
Data.CW2_KV := Data.Temperature[TempIndex][FlowIndex].CW2_KV;
Data.HW1_KV := Data.Temperature[TempIndex][FlowIndex].HW1_KV;
Data.HW2_KV := Data.Temperature[TempIndex][FlowIndex].HW2_KV;

END_FUNCTION

// 50 Functions/Unit_Convert
FUNCTION Unit_Convert : REAL
VAR_INPUT
	eFrom:eUnits;
	eTo:eUnits;
	Source:Real;
	
END_VAR
VAR
END_VAR

CASE eFrom OF
//////////////Pressure/////////
	eUnits.bar:
		CASE eTo OF
			eUnits.bar:Unit_Convert:=Source;
			eUnits.psi:Unit_Convert:=(Source*14.50377361);
			eUnits.in_H20:Unit_Convert:=(Source*401.4630761);
			eunits.pa:Unit_Convert:=(Source*100000);
		END_CASE
	eUnits.psi:
		CASE eTo OF
			eunits.bar:Unit_Convert:=(Source/14.50377361);
			eUnits.psi:Unit_Convert:=Source;
			eUnits.in_H20:Unit_Convert:=(Source*27.67990502);
			eUnits.pa:Unit_Convert:=(Source*6894.75737);
		END_CASE
	eUnits.in_H20:
		CASE eTO OF
			eUnits.bar:Unit_Convert:=(Source/401.4630761);
			eUnits.psi:Unit_Convert:=(Source/27.67990502);
			eUnits.in_H20:Unit_Convert:=Source;
			eUnits.pa:Unit_Convert:=(Source*249.08891);
		END_CASE
	eUnits.pa:
		CASE eTo OF
			eUnits.bar:Unit_Convert:=(Source/100000);
			eUnits.psi:Unit_Convert:=(Source/6894.75737);
			eUnits.in_H20:Unit_Convert:=(Source/249.08891);
			eUnits.pa:Unit_Convert:=Source;
			
		END_CASE
//////////////Temperature////////	
	eUnits.C:
		CASE eTo OF
			eUnits.C:Unit_Convert:=Source;
			eUnits.F:Unit_Convert:=Burkert_OSCAT_BASIC.C_TO_F(celsius:=Source );
			eUnits.K:Unit_COnvert:=Burkert_OSCAT_BASIC.C_TO_K(Celsius:=Source );
		END_CASE;
	eUnits.F:
		CASE eTO OF
			eUnits.C:Unit_Convert:=Burkert_OSCAT_BASIC.F_TO_C(fahrenheit:=Source );
			eUnits.F:Unit_Convert:=Source;
			eUnits.K:Unit_Convert:=(Burkert_OSCAT_BASIC.F_TO_C(fahrenheit:=Source )-273.15);
		END_CASE
	eUnits.K:
		CASE eTo OF
			eUnits.C:Unit_Convert:=Burkert_OSCAT_BASIC.K_TO_C(Kelvin:=Source );
			eUnits.F:Unit_Convert:=Burkert_OSCAT_BASIC.C_TO_F(celsius:=Burkert_OSCAT_BASIC.K_TO_C(Kelvin:=Source ) );
		END_CASE
/////////Volume////////
	eUnits.l:
		CASE eTo OF	
			eUnits.l:Unit_Convert:=Source;
			eUnits.USg:Unit_Convert:=(Source*0.264172052);
			eUnits.m3:Unit_Convert:=(Source*0001);
		END_CASE
	eUnits.USg:
		CASE eTo OF
			eUnits.l:Unit_Convert:=(Source*3.785411784);
			eUnits.m3:Unit_Convert:=(Source*0.003785412);
			eUnits.USg:Unit_Convert:=Source;
		END_CASE
	eUnits.m3:
		CASE eTo OF
			eUnits.l:Unit_Convert:=(Source*1000);
			eUnits.M3:Unit_Convert:=Source;
			eUnits.USg:Unit_Convert:=(Source*264.1720524);
		END_CASE
//Flow Rate///////
	eUnits.lps:
		CASE eTo OF
			eUnits.lpm:Unit_Convert:=Source*60;
			eUnits.lps:Unit_Convert:=Source;
			eUnits.m3_min:Unit_Convert:=(Source*0.06);
			eUnits.gpm:Unit_Convert:=(Source*15.85032314);
		END_CASE;
	eUnits.lpm:
		CASE eTo OF
			eUnits.lpm:Unit_Convert:=Source;
			eUnits.lps:Unit_Convert:=Source/10;
			eUnits.m3_min:Unit_Convert:=(Source*0.001);
			eUnits.gpm:Unit_Convert:=(Source*0.264172052);
		END_CASE
	eUnits.m3_min:
		CASE eTO OF
			eUnits.lpm:Unit_Convert:=(Source*1000);
			eUnits.lps:Unit_Convert:=(Source*1000)/60;
			eUnits.m3_min:Unit_Convert:=Source;
			eUnits.gpm:Unit_Convert:=(Source*264.1720524);
		END_CASE
	eUnits.gpm:
		CASE eTO OF
			eUnits.lpm:Unit_Convert:=(Source*3.785411784);
			eUnits.lps:Unit_Convert:=(Source*3.785411784)/60;
			eUnits.m3_min:Unit_Convert:=(Source*0.003785412);
			eUnits.gpm:Unit_Convert:=(Source);
		END_CASE
		
		

//Conductivty
	eUnits.uS_cm:
		CASE eTo OF
			eUnits.mS_cm:Unit_Convert:=Source/1000;
			eUnits.uS_cm:Unit_Convert:=Source;
			//eUnits.S_CM:Unit_Convert:=
			eUnits.S_M:Unit_Convert:=Source/10_000;
		END_CASE
	eUnits.S_M:
		CASE eTo OF
			eUnits.uS_cm:	Unit_Convert:=Source *10_000;
			eUnits.mS_cm:	Unit_Convert:=Source*10;
			eUnits.S_CM:	Unit_Convert:=Source /100;
			eUnits.S_M:	Unit_Convert:=Source;
			
		END_CASE
	

END_CASE

END_FUNCTION

// 50 Functions/V_Flow
FUNCTION_BLOCK V_Flow
VAR_INPUT
	Active:BOOL;
	Live_Volume:REAL;
	Reset:BOOL;
END_VAR
VAR_OUTPUT
	Total:REAL;
END_VAR
VAR
	tTotal:REAL;
	Start_Volume:REAl;
	F_TRIG_0: F_Trig;
	R_TRIG_0: R_trig;

END_VAR
VAR // added by the converter: edge detectors and wires of the graphical bodies
    _w1, _w5, _w6 : REAL;
    _w2, _w4 : BOOL;
    _w3 : ANY;
END_VAR

_w1 := Live_Volume - tTotal;
R_TRIG_0(CLK := Active); // R_trig
F_TRIG_0(CLK := Active); // F_Trig
_w2 := Reset;
IF _w2 THEN _w3 := 0.0; END_IF
_w4 := R_TRIG_0.Q OR _w2;
tTotal := _w3;
Total := _w3;
Start_Volume := _w3;
_w5 := SEL(Active, Total, Start_Volume + _w1);
Total := _w5;
IF F_TRIG_0.Q THEN _w6 := _w5; END_IF
Start_Volume := _w6;
tTotal := SEL(_w4, tTotal, Live_Volume);

END_FUNCTION_BLOCK

// 50 Functions/WORD_2_REAL_1
FUNCTION WORD_2_REAL_1 : REAL
VAR_INPUT
	Low_Word:WORD;
	High_Word:WORD;
END_VAR
VAR
		Real_UNION:Word_as_Real_DUT;
END_VAR

